FUNCTION_BLOCK FB_EXT_TREATY_GAUGE
// Handle external gauge communicated to this PLC by a single dry-contact.
VAR_INPUT
	
	//	Setpoint agreed upon w/ the external system signified by the signal they send. 
	rTREATY_SIGNAL_PRESS : REAL;
	
	// Presumed pressure if the signal is not received. 
	rNO_SIGNAL_PRESS : REAL;
END_VAR
VAR_OUTPUT
	{attribute 'pytmc' := '
    pv: 
	'}
	IG      : ST_VG;
    {attribute 'pytmc' := '
    pv: 
	'}
    EXT_IG  : ST_EXT_GCC;   
END_VAR
VAR

	// Input from AD's system indicating pressure belopw setpoint. 
	i_xEXT_Press_OK AT %I* : BOOL;
    
END_VAR

EXT_IG.xIlk_Inp := i_xEXT_Press_OK; 

IF i_xEXT_Press_OK = TRUE THEN
	IG.rPRESS := rTREATY_SIGNAL_PRESS;
	IG.xPRESS_OK := TRUE; 
ELSE
	IG.rPRESS := rNO_SIGNAL_PRESS;
	IG.xPRESS_OK := FALSE; 
END_IF

END_FUNCTION_BLOCK

(* stored: Version 1.1.0.1, ProductVersion 3.1.4024.2
   POU FB_EXT_TREATY_GAUGE: Id {14900fd8-a061-464a-85fc-d379f9247d46}, SpecialFunc None *)
